//Converts a RobotPoseSimple to a ARRAY [0..2] OF LREAL
FUNCTION RPS2ARRAY : ARRAY [0..2] OF LREAL
VAR_INPUT
	pose: RobotPoseSimple;
END_VAR
VAR
END_VAR

RPS2ARRAY[0] := pose.x;
RPS2ARRAY[1] := pose.y;
RPS2ARRAY[2] := pose.theta;

END_FUNCTION

(* stored: Version 1.1.0.1, ProductVersion 3.1.4024.11
   POU RPS2ARRAY: Id {300ce0ab-c6c2-43a9-865f-504abeefb5be}, SpecialFunc None *)
